// TIA Portal V20 export
DATA_BLOCK "CONT_C_Clim_DB"   // DB2251
// stored: InstanceOfName CONT_C, OfSystemLibElement CONT_C, OfSystemLibVersion 1.1
CONT_C   // technology object, version 1.1
   // VAR_INPUT
   //    COM_RST : Bool;
   //    MAN_ON : Bool;
   //    PVPER_ON : Bool;
   //    P_SEL : Bool;
   //    I_SEL : Bool;
   //    INT_HOLD : Bool;
   //    I_ITL_ON : Bool;
   //    D_SEL : Bool;
   //    CYCLE : Time;
   //    SP_INT : Real;
   //    PV_IN : Real;
   //    PV_PER : Word;
   //    MAN : Real;
   //    GAIN : Real;
   //    TI : Time;
   //    TD : Time;
   //    TM_LAG : Time;
   //    DEADB_W : Real;
   //    LMN_HLM : Real;
   //    LMN_LLM : Real;
   //    PV_FAC : Real;
   //    PV_OFF : Real;
   //    LMN_FAC : Real;
   //    LMN_OFF : Real;
   //    I_ITLVAL : Real;
   //    DISV : Real;
   // END_VAR
   // VAR_OUTPUT
   //    LMN : Real;
   //    LMN_PER : Word;
   //    QLMN_HLM : Bool;
   //    QLMN_LLM : Bool;
   //    LMN_P : Real;
   //    LMN_I : Real;
   //    LMN_D : Real;
   //    PV : Real;
   //    ER : Real;
   // END_VAR
   // VAR RETAIN
   //    sInvAlt : Real;
   //    sIanteilAlt : Real;
   //    sRestInt : Real;
   //    sRestDif : Real;
   //    sRueck : Real;
   //    sLmn : Real;
   //    sbArwHLmOn : Bool;
   //    sbArwLLmOn : Bool;
   //    sbILimOn : Bool;
   // END_VAR
BEGIN
END_DATA_BLOCK
